# EPICS substitutions: ek9000App/Db/EL1098_mbbiDirect.substitutions
file EL1098.template
{       pattern
        {
                TERMINAL,

        }
        {
        }
}
